Universal Robots PolyScope program: pick_and_place_demo_with_subprograms.urp

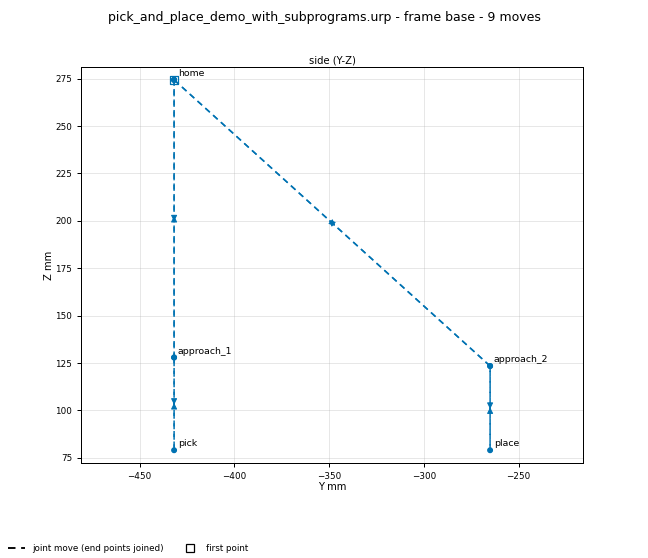
[picture p0: tool path of pick_and_place_demo_with_subprograms.urp in frame base, 9 of 9 moves have a stored position in this frame; points joined in program order, loops and branches not executed]
ProgramRoot setBeforeStartSequence=true; setInitialVariableValues=true; directory=/programs/robotiq_2f_gripper_programs; kinematics=(a=[0, -0.425, -0.39225, 0, 0, 0], d=[0.08916, 0, 0, 0.10915, 0.09465, 0.0823], alpha=[1.5708, 0, 0, 1.5708, -1.5708, 0], deltaTheta=[0, 0, 0, 0, 0, 0], status=notInitialized); name=demo_pick_and_place_with_subprograms; robotEnvironmentFileName=default; serialNumberRobot=2013212154
  InitVariables 
  BeforeStart description=COMMAND_SEQUENCE_BEFORE_PROGRAM_START; name=BeforeStart
    Script type=1; scriptFile=/programs/robotiq_2f_gripper_programs/rq_before_start.script
    Script type=1; scriptFile=/programs/robotiq_2f_gripper_programs/rq_script.script
    Assignment assignmentValueSource=0; expr=0; operatorValueType=INTEGER; valueSource=EXPRESSION; variable=0
    Assignment assignmentValueSource=0; expr=0; operatorValueType=INTEGER; valueSource=EXPRESSION; variable=0
    Assignment assignmentValueSource=0; expr=0; operatorValueType=INTEGER; valueSource=EXPRESSION; variable=0
  MainProgram cartesianAcceleration=1.2; cartesianSpeed=0.25; jointAcceleration=1.3962634015954636; jointSpeed=1.0471975511965976; moveAsFastAsPossible=true; sharedProcessMoveBlendRadius=0.025; featureReference=(installationNameReference=Base); motionType=JOINT_SPACE; runOnlyOneCycle=true
    Comment commentString=This program moves the robot to an object.
    Comment commentString=It then picks it and moves it to another
    Comment commentString=location.
    CallSubProgram subProgramNodeToCall=rq_set_force(rq_force)
    CallSubProgram subProgramNodeToCall=rq_set_speed(rq_speed)
    CallSubProgram subProgramNodeToCall=rq_activate_and_wait()
    CallSubProgram subProgramNodeToCall=rq_open_and_wait()
    Move cartesianAcceleration=1.2; cartesianSpeed=0.25; jointAcceleration=1.3962634015954636; jointSpeed=1.0471975511965976; moveAsFastAsPossible=true; sharedProcessMoveBlendRadius=0.025; featureReference=(installationNameReference=Base); motionType=JOINT_SPACE
      Waypoint blendRadius=0.05; cartesianAcceleration=1.2; cartesianSpeed=0.25; jointAcceleration=1.3962634015954636; jointSpeed=1.0471975511965976; nextMotionTime=2.0; stoppoint=true; useSharedBlendParameter=true; useSharedParameters=true; position=TCP in base x=-120.113 y=-431.761 z=274.386 mm, rx=-0.0012 ry=3.1163 rz=0.0389 rad; joints [-91.713, -87.601, -115.63, -68.242, 91.392, -1.776] deg; positionType=FIXED_POSITION; waypointPoseInFeatureCoordinates=(pos=(x=-0.1201130103353891, y=-0.4317606580015477, z=0.2743855757605886), rot=(x=-0.00122135968159332, y=3.116276528481954, z=0.038891915636889256)); name=home
      Waypoint blendRadius=0.05; cartesianAcceleration=1.2; cartesianSpeed=0.25; jointAcceleration=1.3962634015954636; jointSpeed=1.0471975511965976; nextMotionTime=2.0; stoppoint=true; useSharedBlendParameter=true; useSharedParameters=true; position=TCP in base x=-120.113 y=-431.758 z=127.919 mm, rx=-0.0012 ry=3.1163 rz=0.0389 rad; joints [-91.713, -101.182, -127.255, -43.036, 91.392, -1.776] deg; positionType=FIXED_POSITION; waypointPoseInFeatureCoordinates=(pos=(x=-0.12011292329006278, y=-0.4317577480118261, z=0.12791870504696637), rot=(x=-0.0012213596815903148, y=3.1162765284819804, z=0.03889191563687878)); name=approach_1
    Move cartesianAcceleration=1.2; cartesianSpeed=0.25; jointAcceleration=1.3962634015954636; jointSpeed=1.0471975511965976; moveAsFastAsPossible=true; sharedProcessMoveBlendRadius=0.025; featureReference=(installationNameReference=Base); motionType=JOINT_SPACE
      Waypoint blendRadius=0.05; cartesianAcceleration=1.2; cartesianSpeed=0.25; jointAcceleration=1.3962634015954636; jointSpeed=1.0471975511965976; nextMotionTime=2.0; stoppoint=true; useSharedBlendParameter=true; useSharedParameters=true; position=TCP in base x=-120.113 y=-431.755 z=78.977 mm, rx=-0.0012 ry=3.1163 rz=0.0389 rad; joints [-91.713, -107.888, -129.378, -34.208, 91.392, -1.776] deg; positionType=FIXED_POSITION; waypointPoseInFeatureCoordinates=(pos=(x=-0.12011283734170543, y=-0.4317548746946599, z=0.07897675599398006), rot=(x=-0.0012213596815881583, y=3.1162765284819804, z=0.03889191563688198)); name=pick
      CallSubProgram subProgramNodeToCall=rq_close_and_wait()
      Waypoint blendRadius=0.05; cartesianAcceleration=1.2; cartesianSpeed=0.25; jointAcceleration=1.3962634015954636; jointSpeed=1.0471975511965976; nextMotionTime=2.0; stoppoint=true; useSharedBlendParameter=true; useSharedParameters=true; position=TCP in base x=-120.113 y=-431.758 z=127.919 mm, rx=-0.0012 ry=3.1163 rz=0.0389 rad; joints [-91.713, -101.182, -127.255, -43.036, 91.392, -1.776] deg; positionType=FIXED_POSITION; waypointPoseInFeatureCoordinates=(pos=(x=-0.12011292329006278, y=-0.4317577480118261, z=0.12791870504696637), rot=(x=-0.0012213596815903148, y=3.1162765284819804, z=0.03889191563687878)); name=approach_1
    Move cartesianAcceleration=1.2; cartesianSpeed=0.25; jointAcceleration=1.3962634015954636; jointSpeed=1.0471975511965976; moveAsFastAsPossible=true; sharedProcessMoveBlendRadius=0.025; featureReference=(installationNameReference=Base); motionType=JOINT_SPACE
      Waypoint blendRadius=0.05; cartesianAcceleration=1.2; cartesianSpeed=0.25; jointAcceleration=1.3962634015954636; jointSpeed=1.0471975511965976; nextMotionTime=2.0; stoppoint=true; useSharedBlendParameter=true; useSharedParameters=true; position=TCP in base x=-120.113 y=-431.761 z=274.386 mm, rx=-0.0012 ry=3.1163 rz=0.0389 rad; joints [-91.713, -87.601, -115.63, -68.242, 91.392, -1.776] deg; positionType=FIXED_POSITION; waypointPoseInFeatureCoordinates=(pos=(x=-0.1201130103353891, y=-0.4317606580015477, z=0.2743855757605886), rot=(x=-0.00122135968159332, y=3.116276528481954, z=0.038891915636889256)); name=home
    CallSubProgram subProgramNodeToCall=rq_is_object_detected()
    If expr=ExpressionVariableNode≟0; type=IF_NODE
      Halt 
      Comment commentString=No object detected. Manage the case.
    Move cartesianAcceleration=1.2; cartesianSpeed=0.25; jointAcceleration=1.3962634015954636; jointSpeed=1.0471975511965976; moveAsFastAsPossible=true; sharedProcessMoveBlendRadius=0.025; featureReference=(installationNameReference=Base); motionType=JOINT_SPACE
      Waypoint blendRadius=0.05; cartesianAcceleration=1.2; cartesianSpeed=0.25; jointAcceleration=1.3962634015954636; jointSpeed=1.0471975511965976; nextMotionTime=2.0; stoppoint=true; useSharedBlendParameter=true; useSharedParameters=true; position=TCP in base x=-120.112 y=-265.033 z=123.405 mm, rx=-0.0012 ry=3.1163 rz=0.0389 rad; joints [-92.765, -79.764, -149.961, -41.774, 91.365, -2.827] deg; positionType=FIXED_POSITION; waypointPoseInFeatureCoordinates=(pos=(x=-0.1201119361337282, y=-0.2650331483718448, z=0.12340515561814756), rot=(x=-0.0012213597208201592, y=3.1162765274388784, z=0.038891917212786065)); name=approach_2
    Move cartesianAcceleration=1.2; cartesianSpeed=0.25; jointAcceleration=1.3962634015954636; jointSpeed=1.0471975511965976; moveAsFastAsPossible=true; sharedProcessMoveBlendRadius=0.025; featureReference=(installationNameReference=Base); motionType=JOINT_SPACE
      Waypoint blendRadius=0.05; cartesianAcceleration=1.2; cartesianSpeed=0.25; jointAcceleration=1.3962634015954636; jointSpeed=1.0471975511965976; nextMotionTime=2.0; stoppoint=true; useSharedBlendParameter=true; useSharedParameters=true; position=TCP in base x=-120.112 y=-265.042 z=78.974 mm, rx=-0.0012 ry=3.1163 rz=0.0389 rad; joints [-92.765, -90.253, -153.057, -28.188, 91.365, -2.827] deg; positionType=FIXED_POSITION; waypointPoseInFeatureCoordinates=(pos=(x=-0.12011236076304545, y=-0.2650419420708216, z=0.07897377284993704), rot=(x=-0.001221359720818002, y=3.116276527438878, z=0.0388919172127869)); name=place
      CallSubProgram subProgramNodeToCall=rq_open_and_wait()
      Waypoint blendRadius=0.05; cartesianAcceleration=1.2; cartesianSpeed=0.25; jointAcceleration=1.3962634015954636; jointSpeed=1.0471975511965976; nextMotionTime=2.0; stoppoint=true; useSharedBlendParameter=true; useSharedParameters=true; position=TCP in base x=-120.112 y=-265.033 z=123.405 mm, rx=-0.0012 ry=3.1163 rz=0.0389 rad; joints [-92.765, -79.764, -149.961, -41.774, 91.365, -2.827] deg; positionType=FIXED_POSITION; waypointPoseInFeatureCoordinates=(pos=(x=-0.1201119361337282, y=-0.2650331483718448, z=0.12340515561814756), rot=(x=-0.0012213597208201592, y=3.1162765274388784, z=0.038891917212786065)); name=approach_2
    Move cartesianAcceleration=1.2; cartesianSpeed=0.25; jointAcceleration=1.3962634015954636; jointSpeed=1.0471975511965976; moveAsFastAsPossible=true; sharedProcessMoveBlendRadius=0.025; featureReference=(installationNameReference=Base); motionType=JOINT_SPACE
      Waypoint blendRadius=0.05; cartesianAcceleration=1.2; cartesianSpeed=0.25; jointAcceleration=1.3962634015954636; jointSpeed=1.0471975511965976; nextMotionTime=2.0; stoppoint=true; useSharedBlendParameter=true; useSharedParameters=true; position=TCP in base x=-120.113 y=-431.761 z=274.386 mm, rx=-0.0012 ry=3.1163 rz=0.0389 rad; joints [-91.713, -87.601, -115.63, -68.242, 91.392, -1.776] deg; positionType=FIXED_POSITION; waypointPoseInFeatureCoordinates=(pos=(x=-0.1201130103353891, y=-0.4317606580015477, z=0.2743855757605886), rot=(x=-0.00122135968159332, y=3.116276528481954, z=0.038891915636889256)); name=home
  subProgramToCall [hidden by the author, left out]
  subProgramToCall [hidden by the author, left out]
  subProgramToCall [hidden by the author, left out]
  subProgramToCall [hidden by the author, left out]
  subProgramToCall [hidden by the author, left out]
  subProgramToCall [hidden by the author, left out]
